Fanuc KAREL source: kd00059.KL

-- PROVISIONAL review KL for V940-1; original PC SHA256 6674616f40aae47428c805b1b787fc35e1d5681608d20c7e8369ac44f88702b1
-- Incomplete behavior may be omitted. Consult companion uncertainty JSON. Do not deploy.
PROGRAM KD00059
%NOLOCKGROUP
VAR
  I : INTEGER
  J : INTEGER
  B : BOOLEAN
  R : REAL
  S : STRING[80]
BEGIN
  -- V9_ZERO_TABLE_METADATA_HINT layout=0001; no indexed target words; source/name/runtime held
  -- UNRESOLVED_PC offsets 5-18; opcodes 9D,81,18,9D,1B,9D,12,9C,13,04
  -- UNRESOLVED_PC offsets 23-27; opcodes 7F
END KD00059
